REGION Network 99: SALIDAS - Bajar Mesa Elevadora
   RUNG wire#powerrail
      Contact( #Selec_DW )
      I_Contact( #Selec_UP )
      I_Contact( #Selec_E0_Entrada )
      I_Contact( #Selec_S0_Salida )
      wire#w1
      I_Contact( #MELEV_DW )
      I_Contact( "DB1_SalidasExterioresDeMesa".Mesa[#Mesa].Subir_MElevadora )
      Contact( #EstadoZona.Marcha_CBx )
      I_Contact( #EstadoVI.Error_Mx )
      Coil( "DB1_SalidasExterioresDeMesa".Mesa[#Mesa].Bajar_MElevadora )
   END_RUNG
   RUNG wire#powerrail
      Contact( #Selec_E0_Entrada )
      wire#w2
      Contact( #Pos_E0S0_DW )
      I_Contact( #Pos_E0S0_UP )
      I_Contact( #Selec_DW )
      I_Contact( #Selec_UP )
      I_Contact( #Selec_M1M2_Entrada )
      I_Contact( #Selec_M1M2_Salida )
      I_Contact( #Selec_M3M4_Entrada )
      I_Contact( #Selec_M3M4_Salida )
   END_RUNG wire#w1
   RUNG wire#powerrail
      Contact( #Selec_S0_Salida )
   END_RUNG wire#w2
   RUNG wire#powerrail
      Contact( #Mx_ET01 )
      wire#w3
      I_Contact( #ConfigFB.NoEntrar_E0 )
   END_RUNG wire#w2
   RUNG wire#powerrail
      Contact( #Mx_ET02 )
   END_RUNG wire#w3
   RUNG wire#powerrail
      Contact( #Mx_ET01 )
      Contact( #Pos_Rep_Vacio_DW )
      I_Contact( #Pos_Rep_Vacio_UP )
      wire#w4
      Contact( #ConfigFB.NoEntrar_E0 )
      I_Contact( #Selec_E0_Entrada )
      I_Contact( #Selec_S0_Salida )
      I_Contact( #Selec_DW )
      I_Contact( #Selec_UP )
      I_Contact( #Selec_M1M2_Entrada )
      I_Contact( #Selec_M1M2_Salida )
      I_Contact( #Selec_M3M4_Entrada )
      I_Contact( #Selec_M3M4_Salida )
   END_RUNG wire#w1
   RUNG wire#powerrail
      Contact( #Mx_ET02 )
      Contact( #Pos_Rep_Carga_DW )
      I_Contact( #Pos_Rep_Carga_UP )
   END_RUNG wire#w4
   // the same network as SCL:
   "DB1_SalidasExterioresDeMesa".Mesa[#Mesa].Bajar_MElevadora := ((#Selec_DW AND NOT #Selec_UP AND NOT #Selec_E0_Entrada AND NOT #Selec_S0_Salida) OR ((#Selec_E0_Entrada OR #Selec_S0_Salida OR ((#Mx_ET01 OR #Mx_ET02) AND NOT #ConfigFB.NoEntrar_E0)) AND #Pos_E0S0_DW AND NOT #Pos_E0S0_UP AND NOT #Selec_DW AND NOT #Selec_UP AND NOT #Selec_M1M2_Entrada AND NOT #Selec_M1M2_Salida AND NOT #Selec_M3M4_Entrada AND NOT #Selec_M3M4_Salida) OR (((#Mx_ET01 AND #Pos_Rep_Vacio_DW AND NOT #Pos_Rep_Vacio_UP) OR (#Mx_ET02 AND #Pos_Rep_Carga_DW AND NOT #Pos_Rep_Carga_UP)) AND #ConfigFB.NoEntrar_E0 AND NOT #Selec_E0_Entrada AND NOT #Selec_S0_Salida AND NOT #Selec_DW AND NOT #Selec_UP AND NOT #Selec_M1M2_Entrada AND NOT #Selec_M1M2_Salida AND NOT #Selec_M3M4_Entrada AND NOT #Selec_M3M4_Salida)) AND NOT #MELEV_DW AND NOT "DB1_SalidasExterioresDeMesa".Mesa[#Mesa].Subir_MElevadora AND #EstadoZona.Marcha_CBx AND NOT #EstadoVI.Error_Mx;
END_REGION

REGION Network 100: ESTADOS DE LA MESA
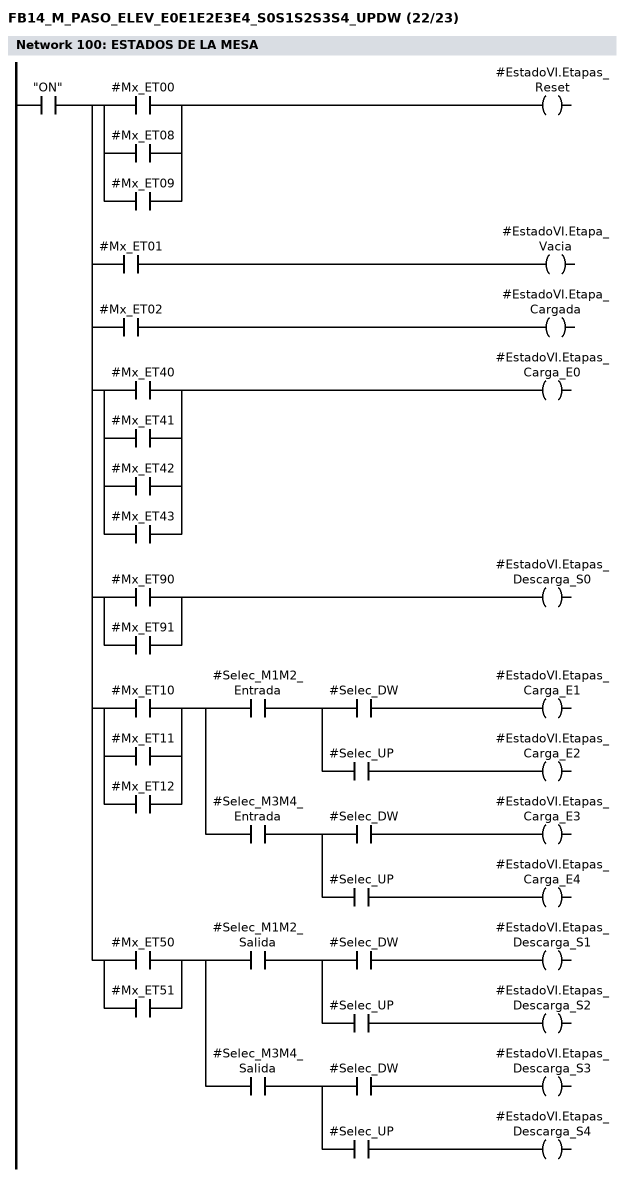
   RUNG wire#powerrail
      Contact( "ON" )
      wire#w1
      Contact( #Mx_ET00 )
      wire#w2
      Coil( #EstadoVI.Etapas_Reset )
   END_RUNG
   RUNG wire#w1
      Contact( #Mx_ET08 )
   END_RUNG wire#w2
   RUNG wire#w1
      Contact( #Mx_ET09 )
   END_RUNG wire#w2
   RUNG wire#w1
      Contact( #Mx_ET01 )
      Coil( #EstadoVI.Etapa_Vacia )
   END_RUNG
   RUNG wire#w1
      Contact( #Mx_ET02 )
      Coil( #EstadoVI.Etapa_Cargada )
   END_RUNG
   RUNG wire#w1
      Contact( #Mx_ET40 )
      wire#w3
      Coil( #EstadoVI.Etapas_Carga_E0 )
   END_RUNG
   RUNG wire#w1
      Contact( #Mx_ET41 )
   END_RUNG wire#w3
   RUNG wire#w1
      Contact( #Mx_ET42 )
   END_RUNG wire#w3
   RUNG wire#w1
      Contact( #Mx_ET43 )
   END_RUNG wire#w3
   RUNG wire#w1
      Contact( #Mx_ET90 )
      wire#w4
      Coil( #EstadoVI.Etapas_Descarga_S0 )
   END_RUNG
   RUNG wire#w1
      Contact( #Mx_ET91 )
   END_RUNG wire#w4
   RUNG wire#w1
      Contact( #Mx_ET10 )
      wire#w5
      Contact( #Selec_M1M2_Entrada )
      wire#w6
      Contact( #Selec_DW )
      Coil( #EstadoVI.Etapas_Carga_E1 )
   END_RUNG
   RUNG wire#w1
      Contact( #Mx_ET11 )
   END_RUNG wire#w5
   RUNG wire#w1
      Contact( #Mx_ET12 )
   END_RUNG wire#w5
   RUNG wire#w6
      Contact( #Selec_UP )
      Coil( #EstadoVI.Etapas_Carga_E2 )
   END_RUNG
   RUNG wire#w5
      Contact( #Selec_M3M4_Entrada )
      wire#w7
      Contact( #Selec_DW )
      Coil( #EstadoVI.Etapas_Carga_E3 )
   END_RUNG
   RUNG wire#w7
      Contact( #Selec_UP )
      Coil( #EstadoVI.Etapas_Carga_E4 )
   END_RUNG
   RUNG wire#w1
      Contact( #Mx_ET50 )
      wire#w8
      Contact( #Selec_M1M2_Salida )
      wire#w9
      Contact( #Selec_DW )
      Coil( #EstadoVI.Etapas_Descarga_S1 )
   END_RUNG
   RUNG wire#w1
      Contact( #Mx_ET51 )
   END_RUNG wire#w8
   RUNG wire#w9
      Contact( #Selec_UP )
      Coil( #EstadoVI.Etapas_Descarga_S2 )
   END_RUNG
   RUNG wire#w8
      Contact( #Selec_M3M4_Salida )
      wire#w10
      Contact( #Selec_DW )
      Coil( #EstadoVI.Etapas_Descarga_S3 )
   END_RUNG
   RUNG wire#w10
      Contact( #Selec_UP )
      Coil( #EstadoVI.Etapas_Descarga_S4 )
   END_RUNG
   // the same network as SCL:
   #EstadoVI.Etapas_Reset := "ON" AND (#Mx_ET00 OR #Mx_ET08 OR #Mx_ET09);
   #EstadoVI.Etapa_Vacia := "ON" AND #Mx_ET01;
   #EstadoVI.Etapa_Cargada := "ON" AND #Mx_ET02;
   #EstadoVI.Etapas_Carga_E0 := "ON" AND (#Mx_ET40 OR #Mx_ET41 OR #Mx_ET42 OR #Mx_ET43);
   #EstadoVI.Etapas_Descarga_S0 := "ON" AND (#Mx_ET90 OR #Mx_ET91);
   #_w1 := "ON" AND (#Mx_ET10 OR #Mx_ET11 OR #Mx_ET12);
   #_w2 := #_w1 AND #Selec_M1M2_Entrada;
   #EstadoVI.Etapas_Carga_E1 := #_w2 AND #Selec_DW;
   #EstadoVI.Etapas_Carga_E2 := #_w2 AND #Selec_UP;
   #_w3 := #_w1 AND #Selec_M3M4_Entrada;
   #EstadoVI.Etapas_Carga_E3 := #_w3 AND #Selec_DW;
   #EstadoVI.Etapas_Carga_E4 := #_w3 AND #Selec_UP;
   #_w4 := "ON" AND (#Mx_ET50 OR #Mx_ET51);
   #_w5 := #_w4 AND #Selec_M1M2_Salida;
   #EstadoVI.Etapas_Descarga_S1 := #_w5 AND #Selec_DW;
   #EstadoVI.Etapas_Descarga_S2 := #_w5 AND #Selec_UP;
   #_w6 := #_w4 AND #Selec_M3M4_Salida;
   #EstadoVI.Etapas_Descarga_S3 := #_w6 AND #Selec_DW;
   #EstadoVI.Etapas_Descarga_S4 := #_w6 AND #Selec_UP;
END_REGION

REGION Network 101: ENTRADAS DE LA MESA
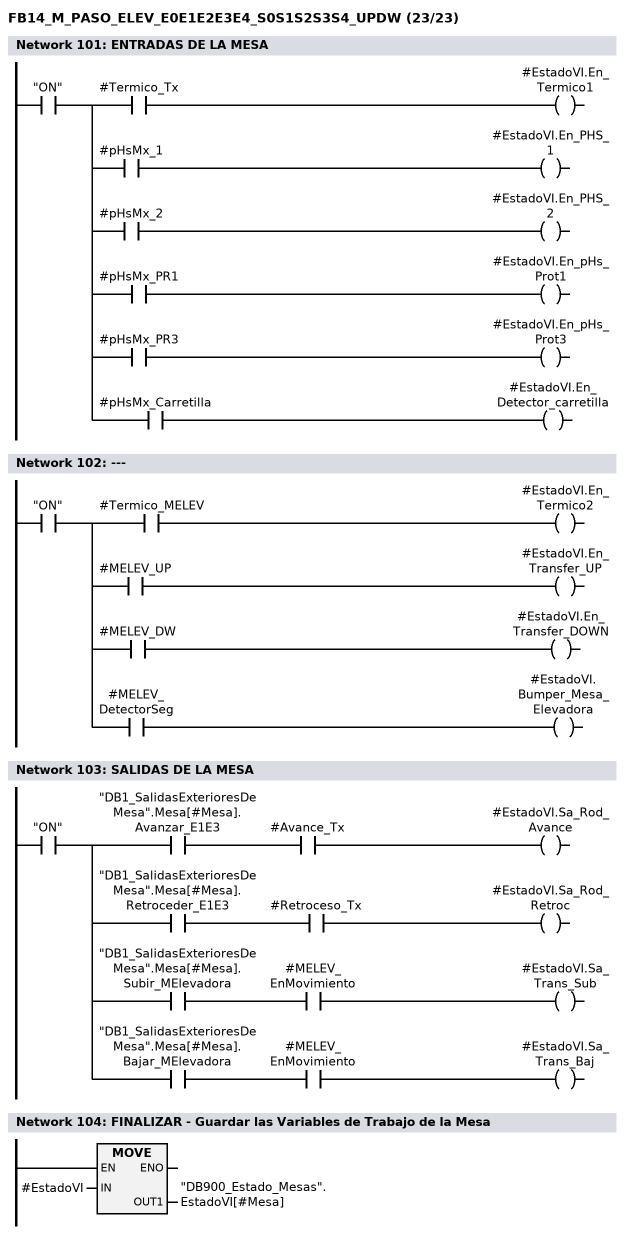
   RUNG wire#powerrail
      Contact( "ON" )
      wire#w1
      Contact( #Termico_Tx )
      Coil( #EstadoVI.En_Termico1 )
   END_RUNG
   RUNG wire#w1
      Contact( #pHsMx_1 )
      Coil( #EstadoVI.En_PHS_1 )
   END_RUNG
   RUNG wire#w1
      Contact( #pHsMx_2 )
      Coil( #EstadoVI.En_PHS_2 )
   END_RUNG
   RUNG wire#w1
      Contact( #pHsMx_PR1 )
      Coil( #EstadoVI.En_pHs_Prot1 )
   END_RUNG
   RUNG wire#w1
      Contact( #pHsMx_PR3 )
      Coil( #EstadoVI.En_pHs_Prot3 )
   END_RUNG
   RUNG wire#w1
      Contact( #pHsMx_Carretilla )
      Coil( #EstadoVI.En_Detector_carretilla )
   END_RUNG
   // the same network as SCL:
   #EstadoVI.En_Termico1 := "ON" AND #Termico_Tx;
   #EstadoVI.En_PHS_1 := "ON" AND #pHsMx_1;
   #EstadoVI.En_PHS_2 := "ON" AND #pHsMx_2;
   #EstadoVI.En_pHs_Prot1 := "ON" AND #pHsMx_PR1;
   #EstadoVI.En_pHs_Prot3 := "ON" AND #pHsMx_PR3;
   #EstadoVI.En_Detector_carretilla := "ON" AND #pHsMx_Carretilla;
END_REGION

REGION Network 102: ---
   RUNG wire#powerrail
      Contact( "ON" )
      wire#w1
      Contact( #Termico_MELEV )
      Coil( #EstadoVI.En_Termico2 )
   END_RUNG
   RUNG wire#w1
      Contact( #MELEV_UP )
      Coil( #EstadoVI.En_Transfer_UP )
   END_RUNG
   RUNG wire#w1
      Contact( #MELEV_DW )
      Coil( #EstadoVI.En_Transfer_DOWN )
   END_RUNG
   RUNG wire#w1
      Contact( #MELEV_DetectorSeg )
      Coil( #EstadoVI.Bumper_Mesa_Elevadora )
   END_RUNG
   // the same network as SCL:
   #EstadoVI.En_Termico2 := "ON" AND #Termico_MELEV;
   #EstadoVI.En_Transfer_UP := "ON" AND #MELEV_UP;
   #EstadoVI.En_Transfer_DOWN := "ON" AND #MELEV_DW;
   #EstadoVI.Bumper_Mesa_Elevadora := "ON" AND #MELEV_DetectorSeg;
END_REGION

REGION Network 103: SALIDAS DE LA MESA
   RUNG wire#powerrail
      Contact( "ON" )
      wire#w1
      Contact( "DB1_SalidasExterioresDeMesa".Mesa[#Mesa].Avanzar_E1E3 )
      Contact( #Avance_Tx )
      Coil( #EstadoVI.Sa_Rod_Avance )
   END_RUNG
   RUNG wire#w1
      Contact( "DB1_SalidasExterioresDeMesa".Mesa[#Mesa].Retroceder_E1E3 )
      Contact( #Retroceso_Tx )
      Coil( #EstadoVI.Sa_Rod_Retroc )
   END_RUNG
   RUNG wire#w1
      Contact( "DB1_SalidasExterioresDeMesa".Mesa[#Mesa].Subir_MElevadora )
      Contact( #MELEV_EnMovimiento )
      Coil( #EstadoVI.Sa_Trans_Sub )
   END_RUNG
   RUNG wire#w1
      Contact( "DB1_SalidasExterioresDeMesa".Mesa[#Mesa].Bajar_MElevadora )
      Contact( #MELEV_EnMovimiento )
      Coil( #EstadoVI.Sa_Trans_Baj )
   END_RUNG
   // the same network as SCL:
   #EstadoVI.Sa_Rod_Avance := "ON" AND "DB1_SalidasExterioresDeMesa".Mesa[#Mesa].Avanzar_E1E3 AND #Avance_Tx;
   #EstadoVI.Sa_Rod_Retroc := "ON" AND "DB1_SalidasExterioresDeMesa".Mesa[#Mesa].Retroceder_E1E3 AND #Retroceso_Tx;
   #EstadoVI.Sa_Trans_Sub := "ON" AND "DB1_SalidasExterioresDeMesa".Mesa[#Mesa].Subir_MElevadora AND #MELEV_EnMovimiento;
   #EstadoVI.Sa_Trans_Baj := "ON" AND "DB1_SalidasExterioresDeMesa".Mesa[#Mesa].Bajar_MElevadora AND #MELEV_EnMovimiento;
END_REGION

REGION Network 104: FINALIZAR - Guardar las Variables de Trabajo de la Mesa
   RUNG wire#powerrail
      Move(in := #EstadoVI, out1 => "DB900_Estado_Mesas".EstadoVI[#Mesa])
   END_RUNG
   // the same network as SCL:
   "DB900_Estado_Mesas".EstadoVI[#Mesa] := #EstadoVI;
END_REGION
END_FUNCTION_BLOCK
